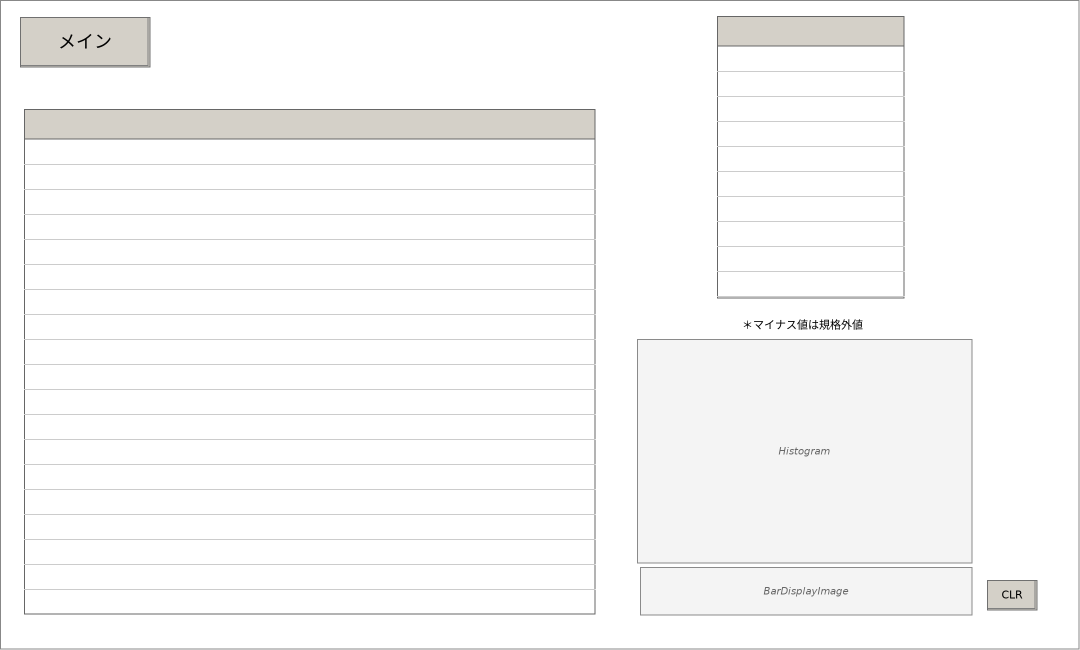
VISUALIZATION s_gateLengthData  // 1080x650
    Rectangle (0,0 1080x650)
        OnMouseClick: change screen: Previous 
    Table (717,16 187x282), data array: gvl_visu.var_gateLengthList
        p3854506369: gvl_visu.var_gateLengthList[INDEX]
        p2232123230: ゲート長さ
    Histogram (637,339 335x224), scale format: %.1f, scale -3..3
        p1518820177: gvl_visu.var_gateLengthList
        p102497268: gvl_visu.var_gateLengthList
        p788070771: ARRAY [0..49] OF REAL
    BarDisplayImage (640,567 332x48), value: gvl_visu.var_curenntGateData, style: BarDisplayImage-Gray, scale format: %.1f, scale 0..3
    Button (20,17 130x50), "メイン"
        OnMouseClick: change screen: s_auto
    Label (739,310 150x30), "＊マイナス値は規格外値"
    Table (24,109 571x505), data array: gvl_visu.var_gateLengthListCav
        p3854506369: gvl_visu.var_gateLengthListCav[1][INDEX]
        p1892666644: gvl_visu.var_gateLengthListCav[2][INDEX]
        p338671338: gvl_visu.var_gateLengthListCav[3][INDEX]
        p2170511999: gvl_visu.var_gateLengthListCav[4][INDEX]
        p3723444502: gvl_visu.var_gateLengthListCav[5][INDEX]
        p1218418051: gvl_visu.var_gateLengthListCav[6][INDEX]
        p746581629: gvl_visu.var_gateLengthListCav[7][INDEX]
        p3104783080: gvl_visu.var_gateLengthListCav[8][INDEX]
        p2232123230: Cav1
        p511219082: Cav2
        p1755163831: Cav3
        p4092479075: Cav4
        p2237128397: Cav5
        p505689113: Cav6
        p1757482276: Cav7
        p4088588272: Cav8
    Button (987,580 50x30), "CLR"
        tap gvl_visu.flg_btn_clrGateData
END_VISUALIZATION

(* stored: Version 1.1.0.1, ProductVersion 3.1.4024.11
   Visu s_gateLengthData: Id {ab0ff8f5-51db-47a5-878e-568794fca185} *)
